(* PLC project Unnamed, Unknown Unnamed 1 *)
(* stored: creationDateTime 2019-08-06T14:23:42, modificationDateTime 2025-04-30T18:17:24 *)

PROGRAM MainStuff
  VAR
    SELECTED_INDEX : HMI_INT := 0;
    SELECTED_INDEX_2 : HMI_INT := 0;
    OPTIONS : HMI_STRING := '5:6:7';
    SELECTED_VALUE : HMI_STRING;
    SELECTED_VALUE_2 : HMI_STRING;
    ADD_BTN : HMI_BOOL;
    NEW_VAL : HMI_INT := 7;
    R_TRIG0 : R_TRIG;
  END_VAR
  VAR  (* added by the conversion: wires and edge detectors of the diagram *)
    _ADD21_ENO : BOOL;
    _ADD21_OUT : HMI_INT;
    _INT_TO_STRING22_ENO : BOOL;
    _INT_TO_STRING22_OUT : STRING;
    _CONCAT4_ENO : BOOL;
    _CONCAT4_OUT : HMI_STRING;
  END_VAR

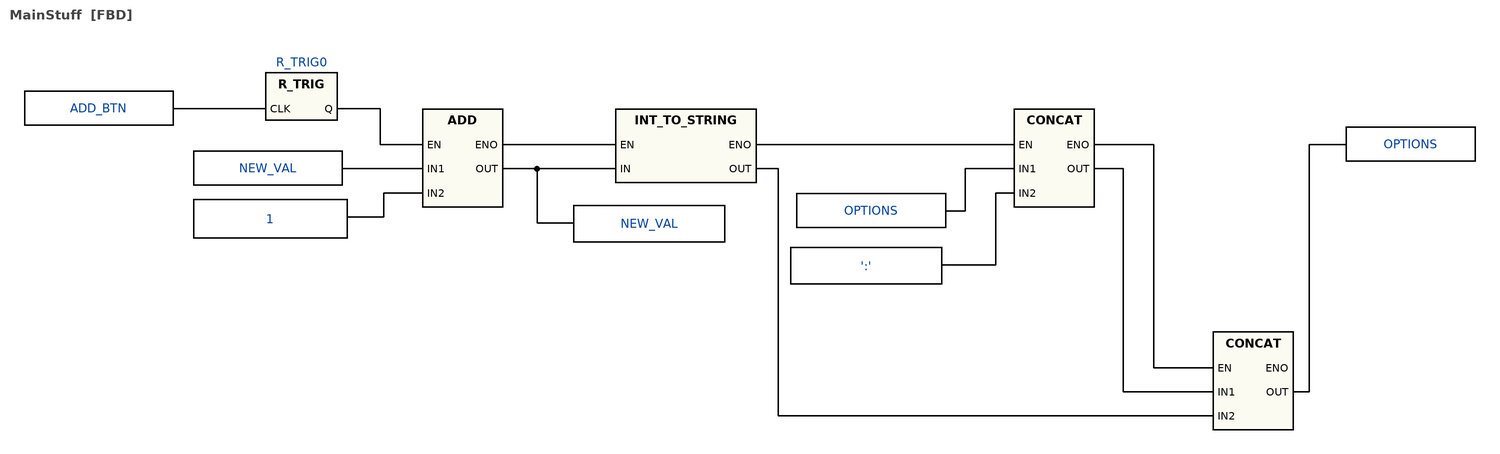
(* FBD diagram, written out as Structured Text *)
R_TRIG0(CLK := ADD_BTN);
_ADD21_OUT := ADD(EN := R_TRIG0.Q, IN1 := NEW_VAL, IN2 := 1, ENO => _ADD21_ENO);
_INT_TO_STRING22_OUT := INT_TO_STRING(EN := _ADD21_ENO, IN := _ADD21_OUT, ENO => _INT_TO_STRING22_ENO);
_CONCAT4_OUT := CONCAT(EN := _INT_TO_STRING22_ENO, IN1 := OPTIONS, IN2 := ':', ENO => _CONCAT4_ENO);
IF _CONCAT4_ENO THEN OPTIONS := CONCAT(_CONCAT4_OUT, _INT_TO_STRING22_OUT); END_IF;
IF _ADD21_ENO THEN NEW_VAL := _ADD21_OUT; END_IF;
END_PROGRAM

CONFIGURATION config
  RESOURCE resource1 ON PLC
    TASK task0(INTERVAL := T#20ms, PRIORITY := 0);
    PROGRAM instance0 WITH task0 : MainStuff;
  END_RESOURCE
END_CONFIGURATION
